{attribute 'qualified_only'}
{attribute 'strict'}
TYPE E_CtrlValveState :
(
	Unknown := 0,
	InPosition := 1,
	Moving := 2,
	Error := -1
);
END_TYPE

(* stored: Version 1.1.0.1, ProductVersion 3.1.4024.12
   DUT E_CtrlValveState: Id {3f49d063-8531-44fe-a097-76b3d7356d5a} *)
